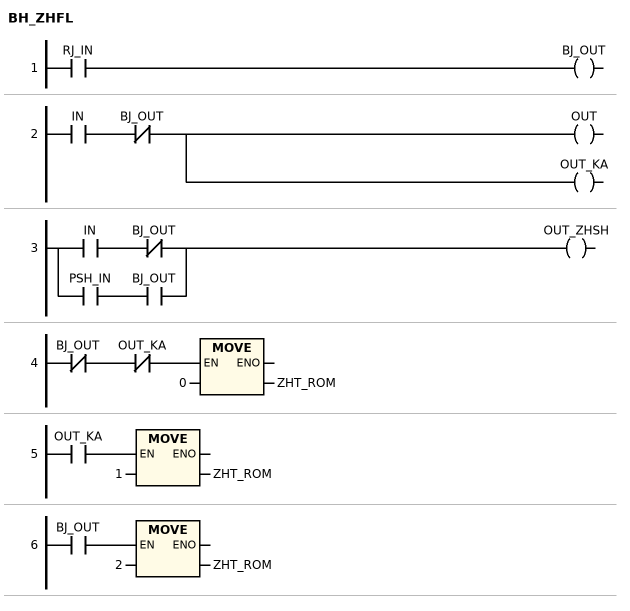
[picture p24: BH_ZHFL (LD)]
_LD_ (* Ladder Diagram *)
NETWORK 1
	[RJ_IN] --- (BJ_OUT)
NETWORK 2
	[IN] - [/BJ_OUT] --- (OUT) (OUT_KA)
NETWORK 3
	{ [IN] - [/BJ_OUT] | [PSH_IN] - [BJ_OUT] } --- (OUT_ZHSH)
NETWORK 4
	[/BJ_OUT] - [/OUT_KA]
		EN --- MOVE(0) => ZHT_ROM
NETWORK 5
	[OUT_KA]
		EN --- MOVE(1) => ZHT_ROM
NETWORK 6
	[BJ_OUT]
		EN --- MOVE(2) => ZHT_ROM
_END_LD_
(* the same logic as Structured Text *)
(* Network 1 *)
BJ_OUT := RJ_IN;
(* Network 2 *)
OUT := IN AND NOT BJ_OUT;
OUT_KA := OUT;
(* Network 3 *)
OUT_ZHSH := IN AND NOT BJ_OUT OR PSH_IN AND BJ_OUT;
(* Network 4 *)
IF NOT BJ_OUT AND NOT OUT_KA THEN
	ZHT_ROM := 0;
END_IF;
(* Network 5 *)
IF OUT_KA THEN
	ZHT_ROM := 1;
END_IF;
(* Network 6 *)
IF BJ_OUT THEN
	ZHT_ROM := 2;
END_IF;
END_FUNCTION_BLOCK

(* POU YOU_FEN, LD *)
FUNCTION_BLOCK YOU_FEN
VAR_INPUT
	MN_IN: INT;
	YW_XZH: INT;
	HIGH_IN: INT;
	LOW_IN: INT;
	YOU_WEI_IN: BOOL;
	TIME_IN: WORD;
	Y_LV_IN: BOOL;
	YL_SET: WORD;

	OPEN_IN: BOOL;
	RESET: BOOL;
	YF_IN: WORD;
	YF_XZ: INT;
END_VAR
VAR_OUTPUT
	YW_XH_OUT: INT;
	YL_KZH: BOOL;
	YOU_WEI_OUT: BOOL;
	TIME_OUT: WORD;
	YL_BJ: BOOL;
	YLV_XH: WORD;
	YL_PT: BOOL;
	YL_OUT: BOOL;
	YF_WD: INT;
	YF_JR: BOOL;
END_VAR
VAR
	TON_YW: YANSHI_OPEN;




	HIGH: BOOL;
	LOW: BOOL;
	KAIJI: BOOL;
	LIMITALARM: LIMITALARM;

	MID_KA: BOOL;
	YLV_YSH: YANSHI_OPEN;
	HYSTERESIS: HYSTERESIS;
	OUT: BOOL;
END_VAR
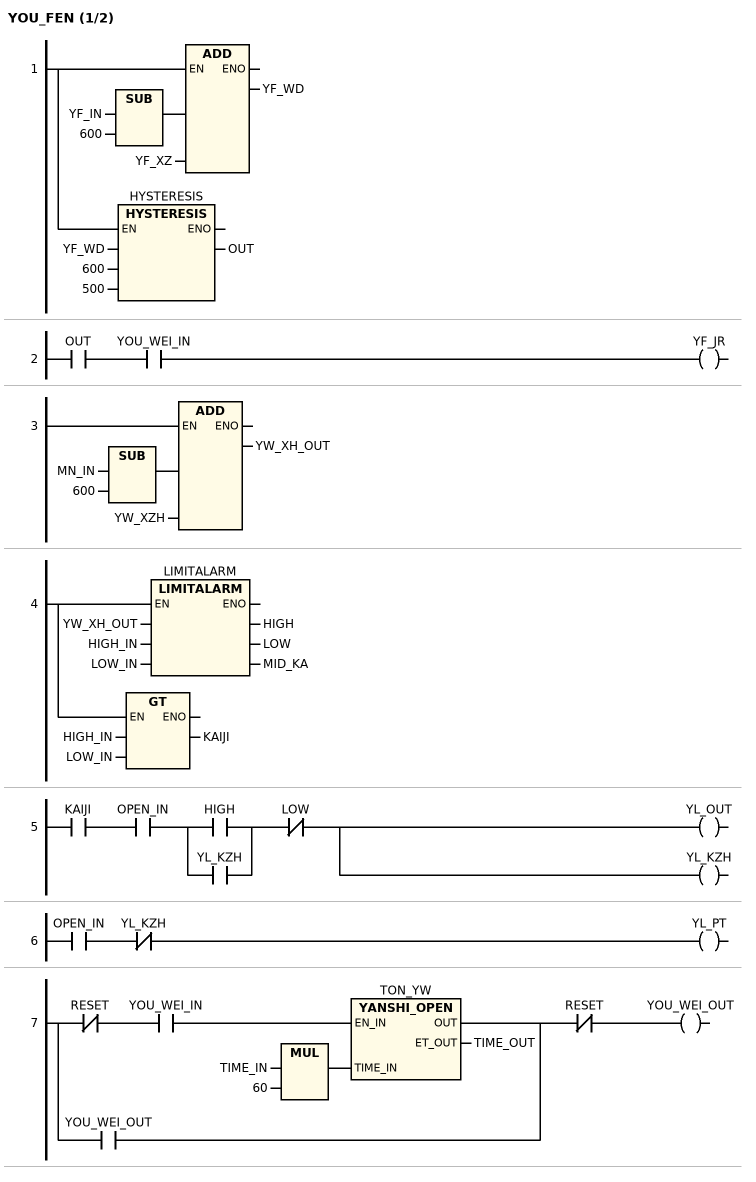
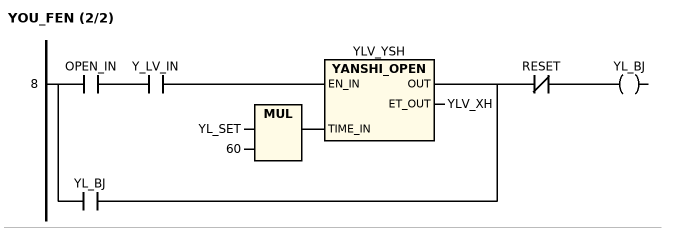
_LD_ (* Ladder Diagram *)
NETWORK 1
	*
		EN --- ADD(SUB(YF_IN, 600), YF_XZ) => YF_WD
		EN --- HYSTERESIS:HYSTERESIS(YF_WD, 600, 500) => OUT
NETWORK 2
	[OUT] - [YOU_WEI_IN] --- (YF_JR)
NETWORK 3
	*
		EN --- ADD(SUB(MN_IN, 600), YW_XZH) => YW_XH_OUT
NETWORK 4
	*
		EN --- LIMITALARM:LIMITALARM(YW_XH_OUT, HIGH_IN, LOW_IN, out 2 => LOW, out 3 => MID_KA) => HIGH
		EN --- GT(HIGH_IN, LOW_IN) => KAIJI
NETWORK 5
	[KAIJI] - [OPEN_IN] - { [HIGH] | [YL_KZH] } - [/LOW] --- (YL_OUT) (YL_KZH)
NETWORK 6
	[OPEN_IN] - [/YL_KZH] --- (YL_PT)
NETWORK 7
	{ [/RESET] - [YOU_WEI_IN] - TON_YW:YANSHI_OPEN(EN_IN: *, TIME_IN: MUL(TIME_IN, 60), ET_OUT => TIME_OUT) | [YOU_WEI_OUT] } - [/RESET] --- (YOU_WEI_OUT)
NETWORK 8
	{ [OPEN_IN] - [Y_LV_IN] - YLV_YSH:YANSHI_OPEN(EN_IN: *, TIME_IN: MUL(YL_SET, 60), ET_OUT => YLV_XH) | [YL_BJ] } - [/RESET] --- (YL_BJ)
_END_LD_
(* the same logic as Structured Text *)
(* Network 1: see the listing above *)
(* Network 2 *)
YF_JR := OUT AND YOU_WEI_IN;
(* Network 3 *)
YW_XH_OUT := (MN_IN - 600) + YW_XZH;
(* Network 4: see the listing above *)
(* Network 5 *)
YL_OUT := KAIJI AND OPEN_IN AND (HIGH OR YL_KZH) AND NOT LOW;
YL_KZH := YL_OUT;
(* Network 6 *)
YL_PT := OPEN_IN AND NOT YL_KZH;
(* Network 7 *)
TON_YW(EN_IN := NOT RESET AND YOU_WEI_IN, TIME_IN := TIME_IN * 60);
TIME_OUT := TON_YW.ET_OUT;
YOU_WEI_OUT := (TON_YW.OUT OR YOU_WEI_OUT) AND NOT RESET;
(* Network 8 *)
YLV_YSH(EN_IN := OPEN_IN AND Y_LV_IN, TIME_IN := YL_SET * 60);
YLV_XH := YLV_YSH.ET_OUT;
YL_BJ := (YLV_YSH.OUT OR YL_BJ) AND NOT RESET;
END_FUNCTION_BLOCK

(* POU SUO, LD *)
FUNCTION_BLOCK SUO
VAR_INPUT
	NIAN_IN: WORD;
	YUE_IN: WORD;
	RI_IN: WORD;
	NIAN_SET_1: WORD;
	YUE_SET_1: WORD;
	RI_SET_1: WORD;
	MIMA_1_IN: WORD;
	MIMA_1_SET_IN: WORD;
	NIAN_SET_2: WORD;
	YUE_SET_2: WORD;
	RI_SET_2: WORD;
	MIMA_2_IN: WORD;
	MIMA_2_SET_IN: WORD;

	NIAN_SET_3: WORD;
	YUE_SET_3: WORD;
	RI_SET_3: WORD;
	MIMA_3_IN: WORD;
	MIMA_3_SET_IN: WORD;
	OFF_ON: BOOL;


END_VAR
VAR_OUTPUT
	SUO_OUT: BOOL;
END_VAR
VAR
	SUO_NIAN_1: BOOL;
	SUO_YUE_1: BOOL;
	SUO_RI_1: BOOL;
	SUO_NIAN_2: BOOL;
	SUO_YUE_2: BOOL;
	SUO_RI_2: BOOL;
	SUO_NIAN_3: BOOL;
	SUO_YUE_3: BOOL;
	SUO_RI_3: BOOL;
	MIMA_1: BOOL;
	MIMA_2: BOOL;
	MIMA_3: BOOL;
	T_SUO_1: TON;
	T_SUO_2: TON;
	T_SUO_3: TON;
	TIME_SUO_1: TIME;
	TIME_SUO_2: TIME;
	TIME_SUO_3: TIME;
END_VAR
VAR_OUTPUT RETAIN
	SUO_1_OUT: BOOL;
	SUO_2_OUT: BOOL;
	SUO_3_OUT: BOOL;
END_VAR
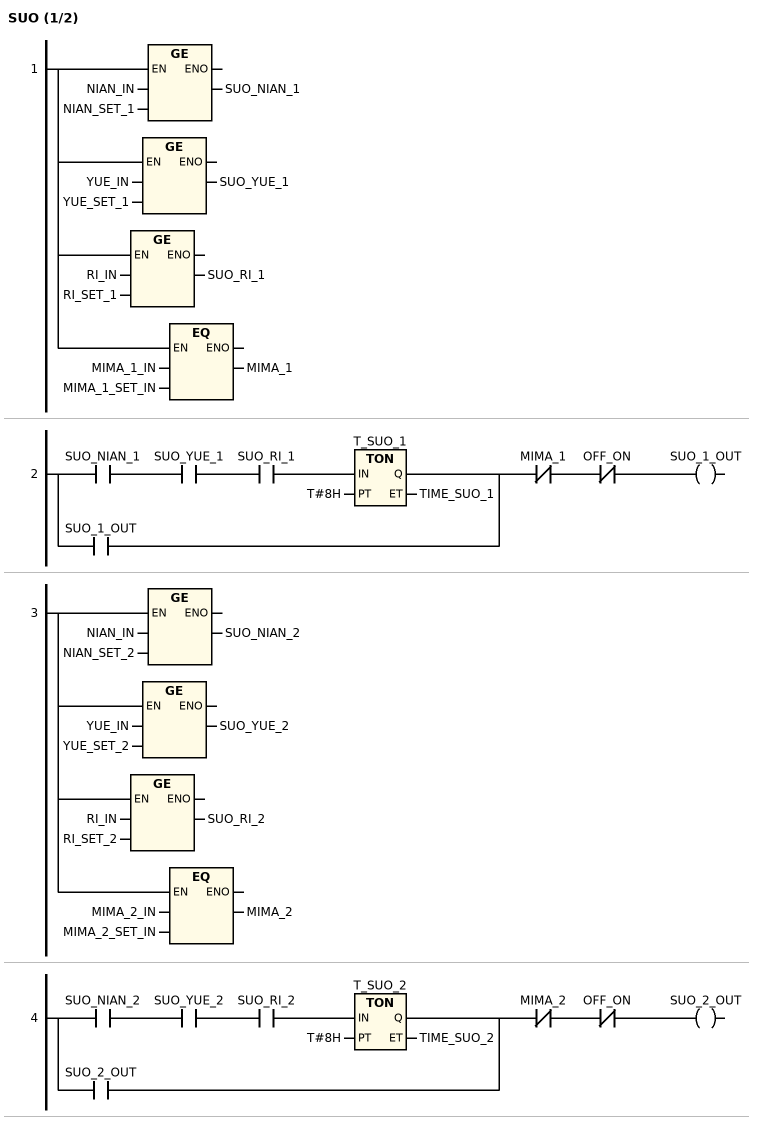
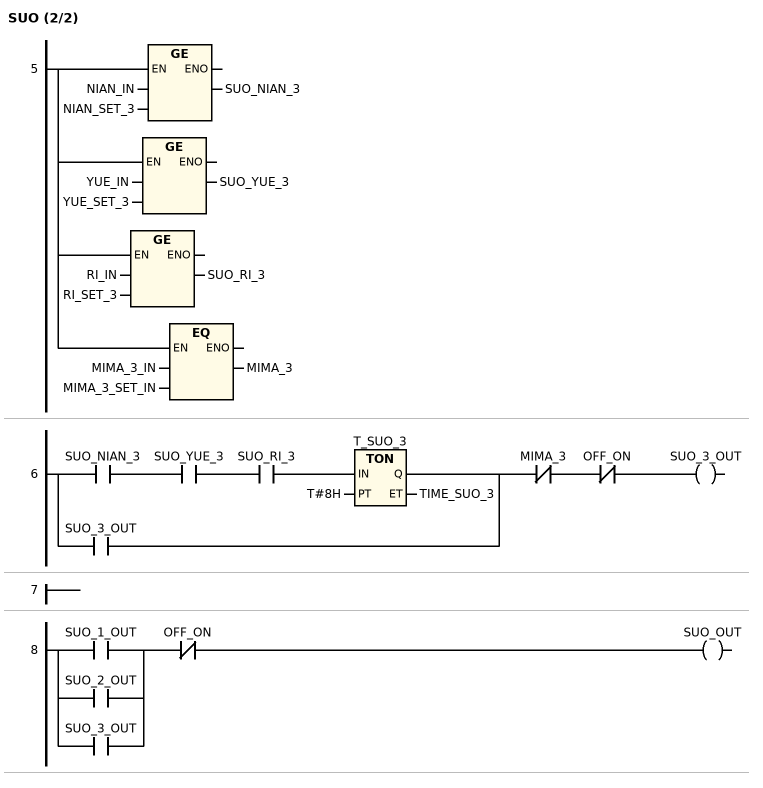
_LD_ (* Ladder Diagram *)
NETWORK 1
	*
		EN --- GE(NIAN_IN, NIAN_SET_1) => SUO_NIAN_1
		EN --- GE(YUE_IN, YUE_SET_1) => SUO_YUE_1
		EN --- GE(RI_IN, RI_SET_1) => SUO_RI_1
		EN --- EQ(MIMA_1_IN, MIMA_1_SET_IN) => MIMA_1
NETWORK 2
	{ [SUO_NIAN_1] - [SUO_YUE_1] - [SUO_RI_1] - T_SUO_1:TON(IN: *, PT: T#8H, ET => TIME_SUO_1) | [SUO_1_OUT] } - [/MIMA_1] - [/OFF_ON] --- (SUO_1_OUT)
NETWORK 3
	*
		EN --- GE(NIAN_IN, NIAN_SET_2) => SUO_NIAN_2
		EN --- GE(YUE_IN, YUE_SET_2) => SUO_YUE_2
		EN --- GE(RI_IN, RI_SET_2) => SUO_RI_2
		EN --- EQ(MIMA_2_IN, MIMA_2_SET_IN) => MIMA_2
NETWORK 4
	{ [SUO_NIAN_2] - [SUO_YUE_2] - [SUO_RI_2] - T_SUO_2:TON(IN: *, PT: T#8H, ET => TIME_SUO_2) | [SUO_2_OUT] } - [/MIMA_2] - [/OFF_ON] --- (SUO_2_OUT)
NETWORK 5
	*
		EN --- GE(NIAN_IN, NIAN_SET_3) => SUO_NIAN_3
		EN --- GE(YUE_IN, YUE_SET_3) => SUO_YUE_3
		EN --- GE(RI_IN, RI_SET_3) => SUO_RI_3
		EN --- EQ(MIMA_3_IN, MIMA_3_SET_IN) => MIMA_3
NETWORK 6
	{ [SUO_NIAN_3] - [SUO_YUE_3] - [SUO_RI_3] - T_SUO_3:TON(IN: *, PT: T#8H, ET => TIME_SUO_3) | [SUO_3_OUT] } - [/MIMA_3] - [/OFF_ON] --- (SUO_3_OUT)
NETWORK 7
	*
NETWORK 8
	{ [SUO_1_OUT] | [SUO_2_OUT] | [SUO_3_OUT] } - [/OFF_ON] --- (SUO_OUT)
_END_LD_
(* the same logic as Structured Text *)
(* Network 1 *)
SUO_NIAN_1 := NIAN_IN >= NIAN_SET_1;
SUO_YUE_1 := YUE_IN >= YUE_SET_1;
SUO_RI_1 := RI_IN >= RI_SET_1;
MIMA_1 := MIMA_1_IN = MIMA_1_SET_IN;
(* Network 2 *)
T_SUO_1(IN := SUO_NIAN_1 AND SUO_YUE_1 AND SUO_RI_1, PT := T#8H);
TIME_SUO_1 := T_SUO_1.ET;
SUO_1_OUT := (T_SUO_1.Q OR SUO_1_OUT) AND NOT MIMA_1 AND NOT OFF_ON;
(* Network 3 *)
SUO_NIAN_2 := NIAN_IN >= NIAN_SET_2;
SUO_YUE_2 := YUE_IN >= YUE_SET_2;
SUO_RI_2 := RI_IN >= RI_SET_2;
MIMA_2 := MIMA_2_IN = MIMA_2_SET_IN;
(* Network 4 *)
T_SUO_2(IN := SUO_NIAN_2 AND SUO_YUE_2 AND SUO_RI_2, PT := T#8H);
TIME_SUO_2 := T_SUO_2.ET;
SUO_2_OUT := (T_SUO_2.Q OR SUO_2_OUT) AND NOT MIMA_2 AND NOT OFF_ON;
(* Network 5 *)
SUO_NIAN_3 := NIAN_IN >= NIAN_SET_3;
SUO_YUE_3 := YUE_IN >= YUE_SET_3;
SUO_RI_3 := RI_IN >= RI_SET_3;
MIMA_3 := MIMA_3_IN = MIMA_3_SET_IN;
(* Network 6 *)
T_SUO_3(IN := SUO_NIAN_3 AND SUO_YUE_3 AND SUO_RI_3, PT := T#8H);
TIME_SUO_3 := T_SUO_3.ET;
SUO_3_OUT := (T_SUO_3.Q OR SUO_3_OUT) AND NOT MIMA_3 AND NOT OFF_ON;
(* Network 7 *)
(* Network 8 *)
SUO_OUT := (SUO_1_OUT OR SUO_2_OUT OR SUO_3_OUT) AND NOT OFF_ON;
END_FUNCTION_BLOCK

(* POU PQ_ZHFL_KZH, LD *)
FUNCTION_BLOCK PQ_ZHFL_KZH
VAR_INPUT
	OPEN_IN: BOOL;
	DY_IN: WORD;
	MNL_XZH: INT;
	DY_MU: INT;
	DY_MD: INT;
	MNL_HIGH_1_IN: INT;
	MNL_LOW_1_IN: INT;
	MNL_HIGH_2_IN: INT;
	MNL_LOW_2_IN: INT;
	MNL_HIGH_3_IN: INT;
	MNL_LOW_3_IN: INT;
	MNL_HIGH_4_IN: INT;
	MNL_LOW_4_IN: INT;
	MNL_HIGH_SHB_IN: INT;
	MNL_LOW_SHB_IN: INT;
	MNL_HIGH_SHB2_IN: INT;
	MNL_LOW_SHB2_IN: INT;
	GY_IN: BOOL;
	LN_AN: BOOL;

	XH_JG: WORD;
	XH_SC: WORD;
	DXJ: BOOL;
	YA_IN: WORD;
	SET_YA: INT;
END_VAR
VAR_OUTPUT
	MNL_OUT: INT;
	FAN_1_OUT: BOOL;
	FAN_2_OUT: BOOL;
	FAN_3_OUT: BOOL;
	FAN_4_OUT: BOOL;
	SHB_OUT: BOOL;
	SHB2_OUT: BOOL;
	LN_NIU: BOOL;
	YOU_YA: INT;
	YA_CHA: INT;
	YA_BJ: BOOL;
END_VAR
VAR
	MNL_R: REAL;
	DIYA: HEX_ENGIN;





	MN_FAN_1: LIMITALARM;
	HIGH_1: BOOL;
	LOW_1: BOOL;
	MID_1: BOOL;
	KAIJI_1: BOOL;
	MN_FAN_2: LIMITALARM;
	HIGH_2: BOOL;
	LOW_2: BOOL;
	MID_2: BOOL;
	KAIJI_2: BOOL;
	MN_FAN_3: LIMITALARM;
	HIGH_3: BOOL;
	LOW_3: BOOL;
	MID_3: BOOL;
	KAIJI_3: BOOL;
	MN_FAN_4: LIMITALARM;
	HIGH_4: BOOL;
	LOW_4: BOOL;
	MID_4: BOOL;
	KAIJI_4: BOOL;
	MN_SHB: LIMITALARM;
	HIGH_SHB: BOOL;
	LOW_SHB: BOOL;
	MID_SHB: BOOL;
	KAIJI_SHB: BOOL;
	MN_SHB2: LIMITALARM;
	HIGH_SHB2: BOOL;
	LOW_SHB2: BOOL;
	MID_SHB2: BOOL;
	KAIJI_SHB2: BOOL;
	ZHFL_KZH: BOOL;
	LN_KZH: AN_NIU;

	BLINK: BLINK;
	DJ_K: BOOL;
	JG_O: BOOL;
	SC_O: BOOL;
	HEX_E: HEX_ENGIN;
END_VAR
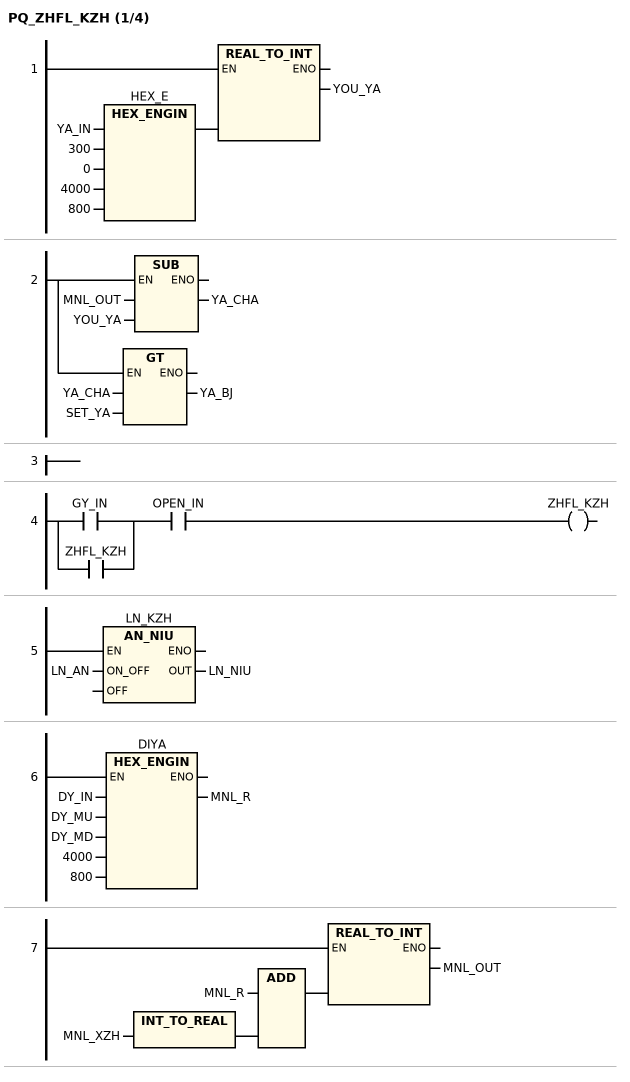
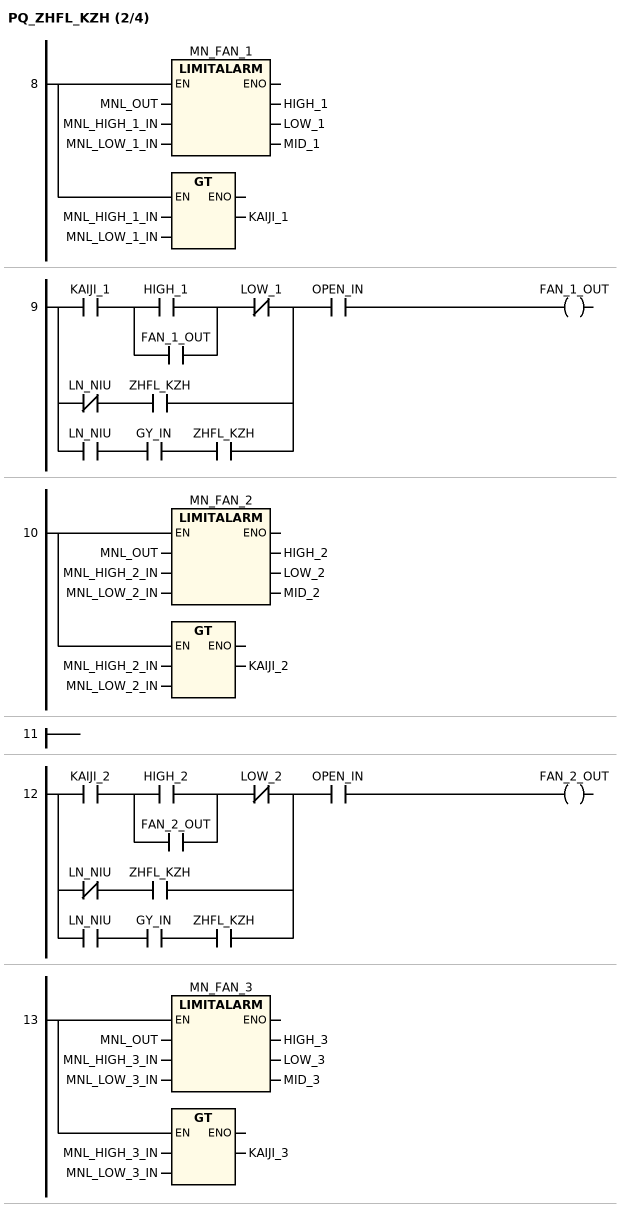
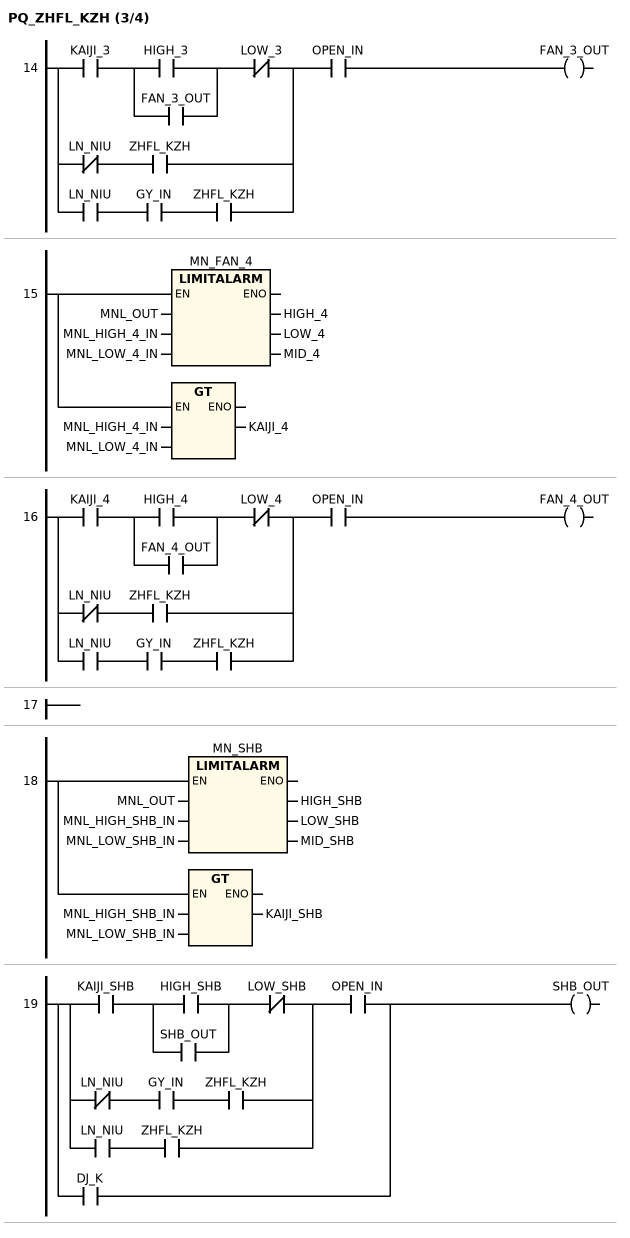
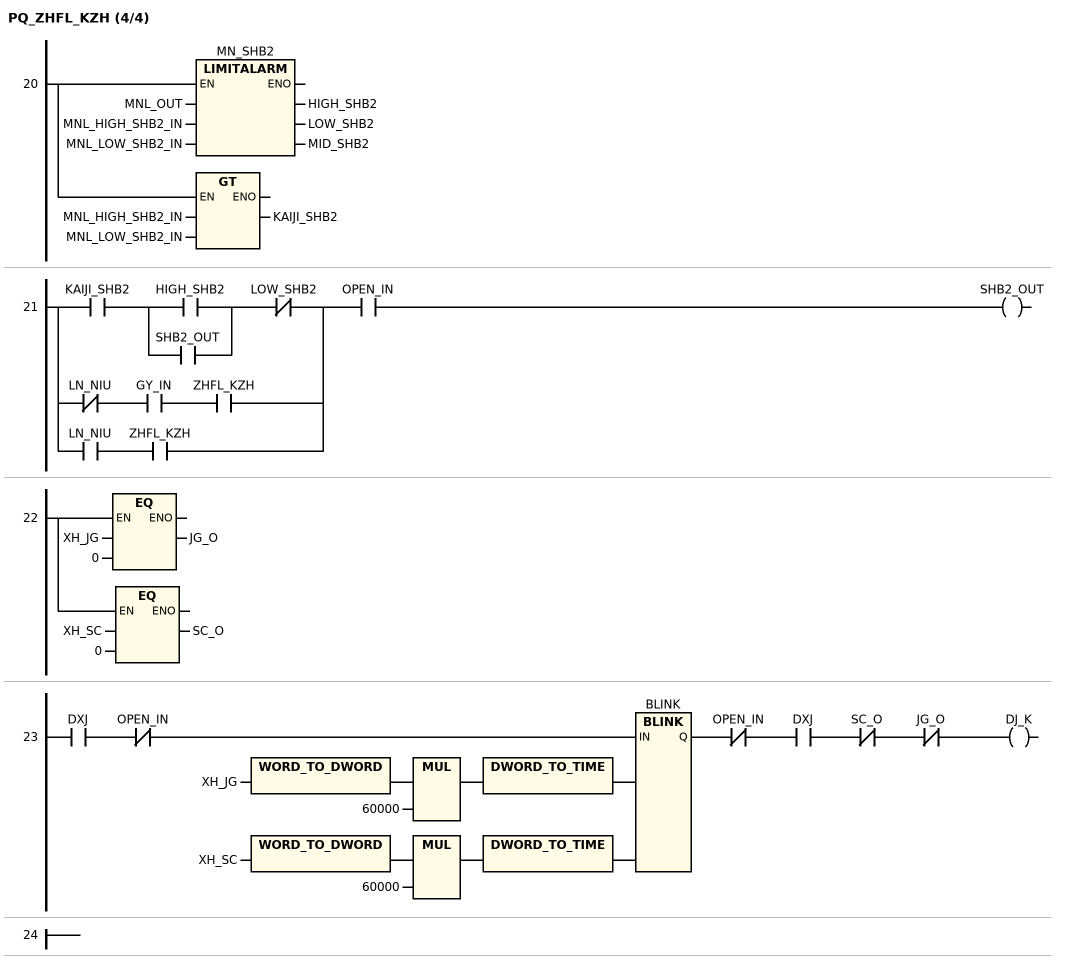
_LD_ (* Ladder Diagram *)
NETWORK 1
	*
		EN --- REAL_TO_INT(HEX_E:HEX_ENGIN(YA_IN, 300, 0, 4000, 800)) => YOU_YA
NETWORK 2
	*
		EN --- SUB(MNL_OUT, YOU_YA) => YA_CHA
		EN --- GT(YA_CHA, SET_YA) => YA_BJ
NETWORK 3
	*
NETWORK 4
	{ [GY_IN] | [ZHFL_KZH] } - [OPEN_IN] --- (ZHFL_KZH)
NETWORK 5
	*
		EN --- LN_KZH:AN_NIU(ON_OFF: LN_AN, OFF: ) => LN_NIU
NETWORK 6
	*
		EN --- DIYA:HEX_ENGIN(DY_IN, DY_MU, DY_MD, 4000, 800) => MNL_R
NETWORK 7
	*
		EN --- REAL_TO_INT(ADD(MNL_R, INT_TO_REAL(MNL_XZH))) => MNL_OUT
NETWORK 8
	*
		EN --- MN_FAN_1:LIMITALARM(MNL_OUT, MNL_HIGH_1_IN, MNL_LOW_1_IN, out 2 => LOW_1, out 3 => MID_1) => HIGH_1
		EN --- GT(MNL_HIGH_1_IN, MNL_LOW_1_IN) => KAIJI_1
NETWORK 9
	{ [KAIJI_1] - { [HIGH_1] | [FAN_1_OUT] } - [/LOW_1] | [/LN_NIU] - [ZHFL_KZH] | [LN_NIU] - [GY_IN] - [ZHFL_KZH] } - [OPEN_IN] --- (FAN_1_OUT)
NETWORK 10
	*
		EN --- MN_FAN_2:LIMITALARM(MNL_OUT, MNL_HIGH_2_IN, MNL_LOW_2_IN, out 2 => LOW_2, out 3 => MID_2) => HIGH_2
		EN --- GT(MNL_HIGH_2_IN, MNL_LOW_2_IN) => KAIJI_2
NETWORK 11
	*
NETWORK 12
	{ [KAIJI_2] - { [HIGH_2] | [FAN_2_OUT] } - [/LOW_2] | [/LN_NIU] - [ZHFL_KZH] | [LN_NIU] - [GY_IN] - [ZHFL_KZH] } - [OPEN_IN] --- (FAN_2_OUT)
NETWORK 13
	*
		EN --- MN_FAN_3:LIMITALARM(MNL_OUT, MNL_HIGH_3_IN, MNL_LOW_3_IN, out 2 => LOW_3, out 3 => MID_3) => HIGH_3
		EN --- GT(MNL_HIGH_3_IN, MNL_LOW_3_IN) => KAIJI_3
NETWORK 14
	{ [KAIJI_3] - { [HIGH_3] | [FAN_3_OUT] } - [/LOW_3] | [/LN_NIU] - [ZHFL_KZH] | [LN_NIU] - [GY_IN] - [ZHFL_KZH] } - [OPEN_IN] --- (FAN_3_OUT)
NETWORK 15
	*
		EN --- MN_FAN_4:LIMITALARM(MNL_OUT, MNL_HIGH_4_IN, MNL_LOW_4_IN, out 2 => LOW_4, out 3 => MID_4) => HIGH_4
		EN --- GT(MNL_HIGH_4_IN, MNL_LOW_4_IN) => KAIJI_4
NETWORK 16
	{ [KAIJI_4] - { [HIGH_4] | [FAN_4_OUT] } - [/LOW_4] | [/LN_NIU] - [ZHFL_KZH] | [LN_NIU] - [GY_IN] - [ZHFL_KZH] } - [OPEN_IN] --- (FAN_4_OUT)
NETWORK 17
	*
NETWORK 18
	*
		EN --- MN_SHB:LIMITALARM(MNL_OUT, MNL_HIGH_SHB_IN, MNL_LOW_SHB_IN, out 2 => LOW_SHB, out 3 => MID_SHB) => HIGH_SHB
		EN --- GT(MNL_HIGH_SHB_IN, MNL_LOW_SHB_IN) => KAIJI_SHB
NETWORK 19
	{ { [KAIJI_SHB] - { [HIGH_SHB] | [SHB_OUT] } - [/LOW_SHB] | [/LN_NIU] - [GY_IN] - [ZHFL_KZH] | [LN_NIU] - [ZHFL_KZH] } - [OPEN_IN] | [DJ_K] } --- (SHB_OUT)
NETWORK 20
	*
		EN --- MN_SHB2:LIMITALARM(MNL_OUT, MNL_HIGH_SHB2_IN, MNL_LOW_SHB2_IN, out 2 => LOW_SHB2, out 3 => MID_SHB2) => HIGH_SHB2
		EN --- GT(MNL_HIGH_SHB2_IN, MNL_LOW_SHB2_IN) => KAIJI_SHB2
NETWORK 21
	{ [KAIJI_SHB2] - { [HIGH_SHB2] | [SHB2_OUT] } - [/LOW_SHB2] | [/LN_NIU] - [GY_IN] - [ZHFL_KZH] | [LN_NIU] - [ZHFL_KZH] } - [OPEN_IN] --- (SHB2_OUT)
NETWORK 22
	*
		EN --- EQ(XH_JG, 0) => JG_O
		EN --- EQ(XH_SC, 0) => SC_O
NETWORK 23
	[DXJ] - [/OPEN_IN] - BLINK:BLINK(*, DWORD_TO_TIME(MUL(WORD_TO_DWORD(XH_JG), 60000)), DWORD_TO_TIME(MUL(WORD_TO_DWORD(XH_SC), 60000))) - [/OPEN_IN] - [DXJ] - [/SC_O] - [/JG_O] --- (DJ_K)
NETWORK 24
	*
_END_LD_
(* the same logic as Structured Text *)
(* Network 1: see the listing above *)
(* Network 2 *)
YA_CHA := MNL_OUT - YOU_YA;
YA_BJ := YA_CHA > SET_YA;
(* Network 3: see the listing above *)
(* Network 4 *)
ZHFL_KZH := (GY_IN OR ZHFL_KZH) AND OPEN_IN;
(* Network 5: see the listing above *)
(* Network 6: see the listing above *)
(* Network 7 *)
MNL_OUT := REAL_TO_INT(MNL_R + INT_TO_REAL(MNL_XZH));
(* Network 8: see the listing above *)
(* Network 9 *)
FAN_1_OUT := (KAIJI_1 AND (HIGH_1 OR FAN_1_OUT) AND NOT LOW_1 OR NOT LN_NIU AND ZHFL_KZH OR LN_NIU AND GY_IN AND ZHFL_KZH) AND OPEN_IN;
(* Network 10: see the listing above *)
(* Network 11: see the listing above *)
(* Network 12 *)
FAN_2_OUT := (KAIJI_2 AND (HIGH_2 OR FAN_2_OUT) AND NOT LOW_2 OR NOT LN_NIU AND ZHFL_KZH OR LN_NIU AND GY_IN AND ZHFL_KZH) AND OPEN_IN;
(* Network 13: see the listing above *)
(* Network 14 *)
FAN_3_OUT := (KAIJI_3 AND (HIGH_3 OR FAN_3_OUT) AND NOT LOW_3 OR NOT LN_NIU AND ZHFL_KZH OR LN_NIU AND GY_IN AND ZHFL_KZH) AND OPEN_IN;
(* Network 15: see the listing above *)
(* Network 16 *)
FAN_4_OUT := (KAIJI_4 AND (HIGH_4 OR FAN_4_OUT) AND NOT LOW_4 OR NOT LN_NIU AND ZHFL_KZH OR LN_NIU AND GY_IN AND ZHFL_KZH) AND OPEN_IN;
(* Network 17: see the listing above *)
(* Network 18: see the listing above *)
(* Network 19 *)
SHB_OUT := (KAIJI_SHB AND (HIGH_SHB OR SHB_OUT) AND NOT LOW_SHB OR NOT LN_NIU AND GY_IN AND ZHFL_KZH OR LN_NIU AND ZHFL_KZH) AND OPEN_IN OR DJ_K;
(* Network 20: see the listing above *)
(* Network 21 *)
SHB2_OUT := (KAIJI_SHB2 AND (HIGH_SHB2 OR SHB2_OUT) AND NOT LOW_SHB2 OR NOT LN_NIU AND GY_IN AND ZHFL_KZH OR LN_NIU AND ZHFL_KZH) AND OPEN_IN;
(* Network 22 *)
JG_O := XH_JG = 0;
SC_O := XH_SC = 0;
(* Network 23: see the listing above *)
(* Network 24: see the listing above *)
END_FUNCTION_BLOCK

(* POU AN_NIU, LD *)
FUNCTION_BLOCK AN_NIU
VAR_INPUT
	ON_OFF: BOOL;
	OFF: BOOL;
END_VAR
VAR_OUTPUT
       END_VAR
VAR
	R1: R_TRIG;
	R1_Q: BOOL;
END_VAR
VAR_OUTPUT RETAIN
	OUT: BOOL;
END_VAR
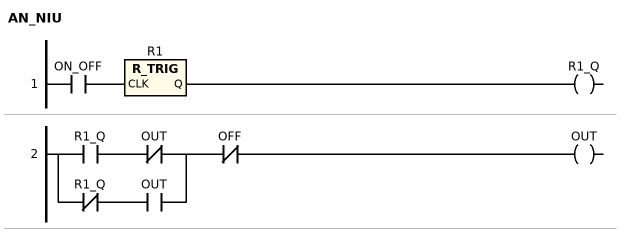
_LD_ (* Ladder Diagram *)
NETWORK 1
	[ON_OFF] - R1:R_TRIG(CLK: *) --- (R1_Q)
NETWORK 2
	{ [R1_Q] - [/OUT] | [/R1_Q] - [OUT] } - [/OFF] --- (OUT)
_END_LD_
(* the same logic as Structured Text *)
(* Network 1 *)
R1(CLK := ON_OFF);
R1_Q := R1.Q;
(* Network 2 *)
OUT := (R1_Q AND NOT OUT OR NOT R1_Q AND OUT) AND NOT OFF;
END_FUNCTION_BLOCK

(* POU XH_YANSHI_1, LD *)
FUNCTION_BLOCK XH_YANSHI_1
VAR_INPUT
	WBKZL_IN: BOOL;
	OPEN_IN: BOOL;
	DY_IN: WORD;
	MNL_XZH: INT;
	MNL_HIGH_IN: INT;
	MNL_LOW_IN: INT;
	OPEN_YSH: WORD;
	CLOSE_YSH: WORD;
	JQ_OPEN_YSH: WORD;
 	JQ_1_BH_IN: BOOL;
	JQ_2_BH_IN: BOOL;
	JQ_3_BH_IN: BOOL;
	JQ_4_BH_IN: BOOL;
	JQ_5_BH_IN: BOOL;
	JQ_6_BH_IN: BOOL;


	DY_MU: INT;
	DY_MD: INT;
	JQ_NJ_SHU: WORD;
	WD_IN: WORD;
	XQ_WD_XZH: INT;
	WD_MU: INT;
	WD_MD: INT;
	GRD_IN: INT;
	GRD_YSH_SET: WORD;
	TD_R: BOOL;
	TJ_ZHH: BOOL;

	YSJ_IN: BOOL;
	RESET: BOOL;
END_VAR
VAR_OUTPUT
	MNL_OUT: INT;
	YL_T_OUT: INT;
	XH_T_XSH: WORD;
	XH_SHU_OUT: WORD;
	XH_ZHT: WORD;


	JJQ_OUT: BOOL;
	XQ_WD_OUT: INT;
	GRD_OUT: INT;
	GRD_ALA: BOOL;
	GRD_YSH_XSH: WORD;
	TJ_ZHH_OUT: BOOL;
END_VAR
VAR
	HIGH: BOOL;
	MID: BOOL;
	CLOSE_SET: TIME;
	OPEN_SET: TIME;
	JQ_OPEN_SET: TIME;
	H_R_Q: BOOL;
	H_TON: TON;
	JT_TON: TON;
	JT_KA: BOOL;
	XH_JD: BOOL;
	JT_SHU: WORD;
	XH_STOP: BOOL;
	XH_NE_3: BOOL;
	JQ_A_OPEN_SET_0: BOOL;
	LOW_R: R_TRIG;
	LOW_R_Q: BOOL;
	L_R_Q: BOOL;
	L_TON: TON;
	XH_SHU_0: BOOL;
	JQ_OPEN_SET_0: BOOL;
	LOW: BOOL;
	XH_NE_6: BOOL;
	XH_NE_12: BOOL;
	XH_NE_18: BOOL;
	XH_EQ_3: BOOL;
	XH_EQ_6: BOOL;
	XH_EQ_9: BOOL;
	XH_EQ_12: BOOL;
	XH_EQ_15: BOOL;
	XH_EQ_18: BOOL;
	HIG_R: R_TRIG;
	XH_NE_9: BOOL;
	MNL_R: REAL;
	MONI_LIANG: LIMITALARM;
	HIGH_KA: BOOL;
	LOW_KA: BOOL;
	MID_KA: BOOL;
	KAIJI: BOOL;
	XH_SHU: WORD;
	OPEN_ET: TIME;
	CLOSE_ET: TIME;
	JT_OPEN_ET: TIME;
	XH_JT_KA: BOOL;
	HIG_KA_R: R_TRIG;
	DIYA: HEX_ENGIN;
	YL_WD: YL_WD;



	MID_R: R_TRIG;


	GRD_KA: BOOL;
	GRD_OPEN: YANSHI_OPEN;
	GRD_KA_0: BOOL;
	JQ_NJ_SHU_0: BOOL;
	JJQ_TOF: TOF;
	TJ_AN: AN_NIU;
	HEX_ENGIN: HEX_ENGIN;
	wd: HEX_ENGIN;
	HEX_ENGI: HEX_ENGIN;
	XW: INT;
END_VAR
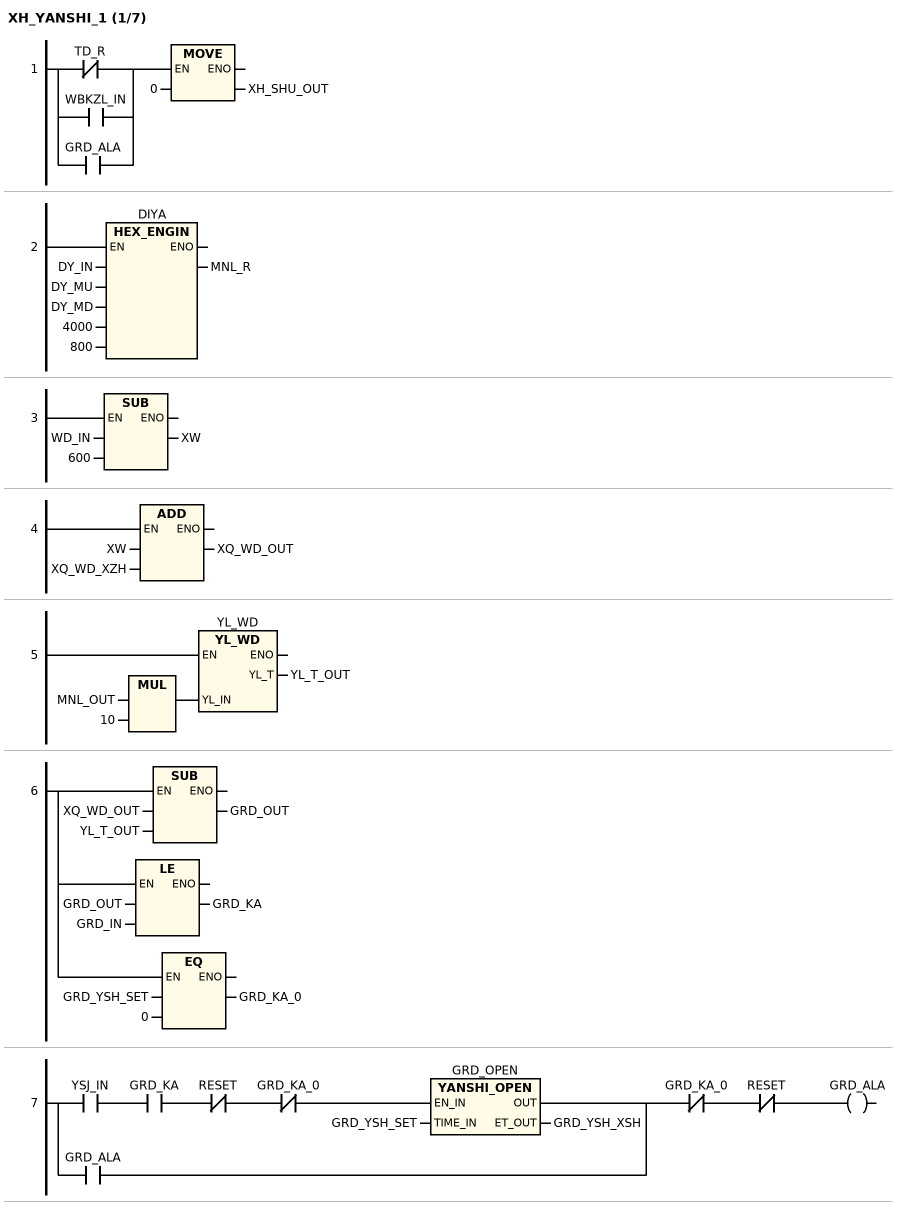
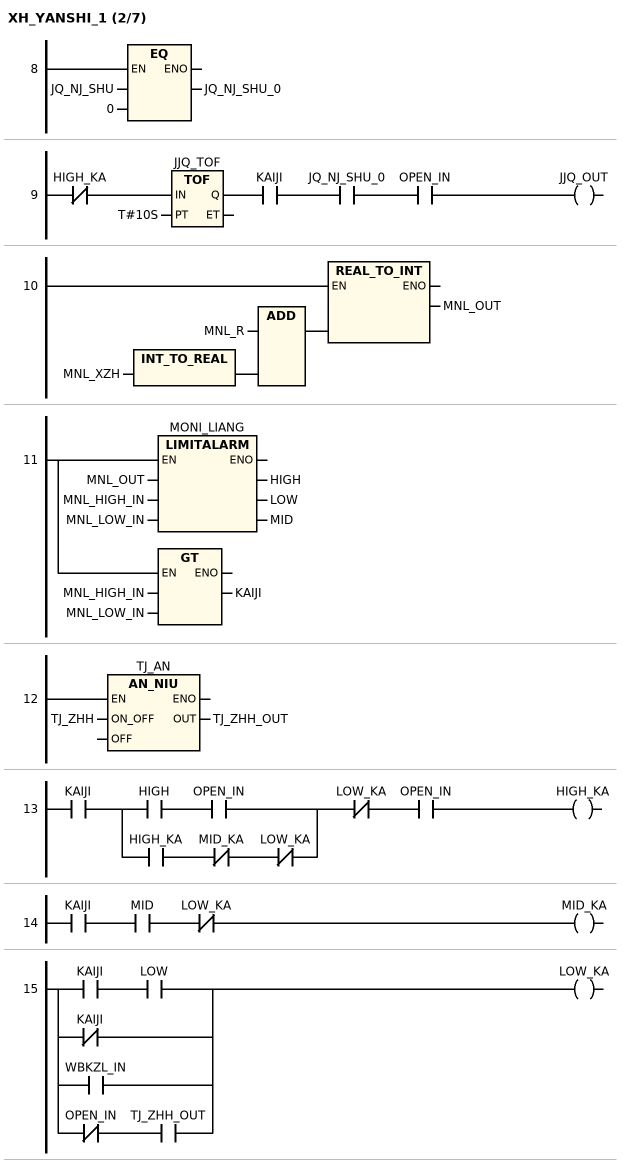
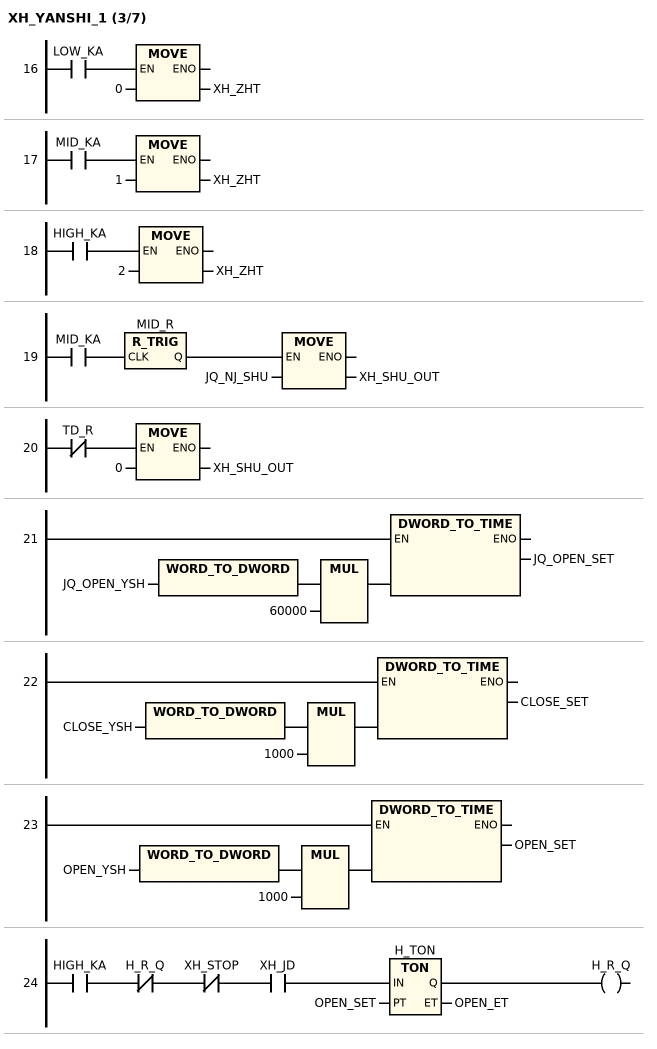
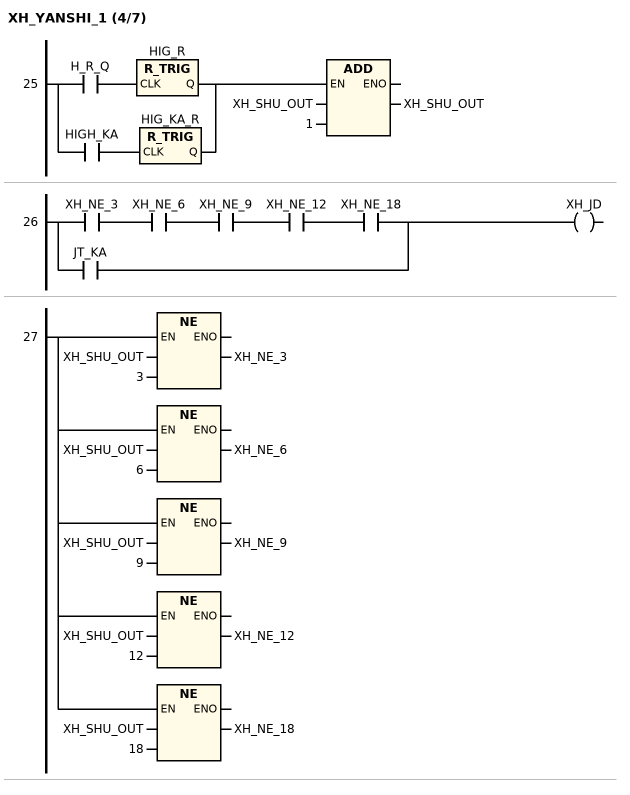
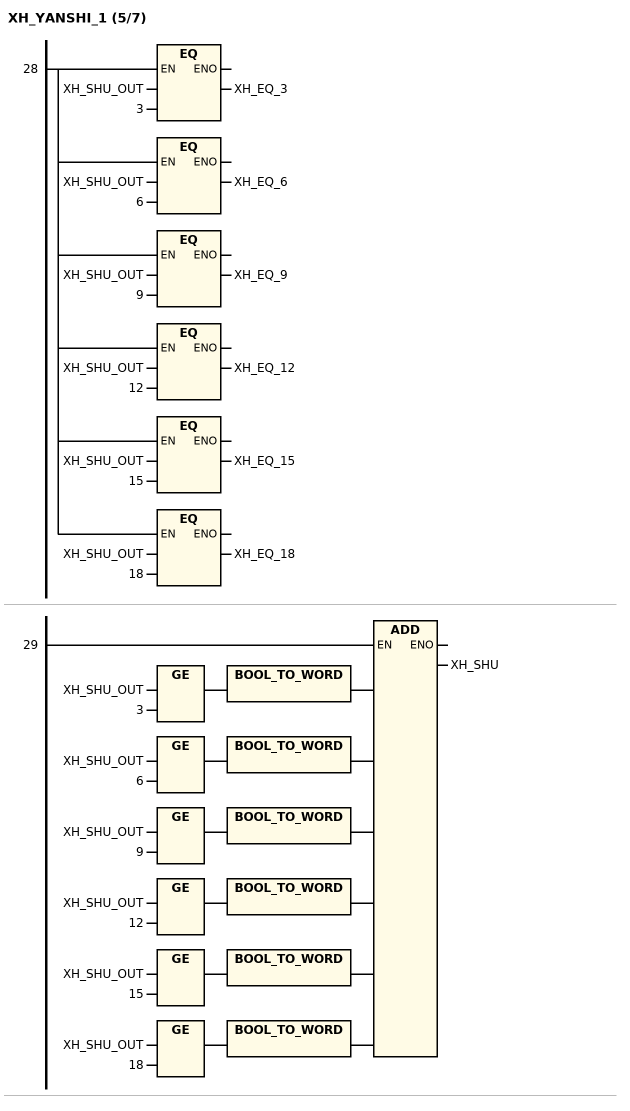
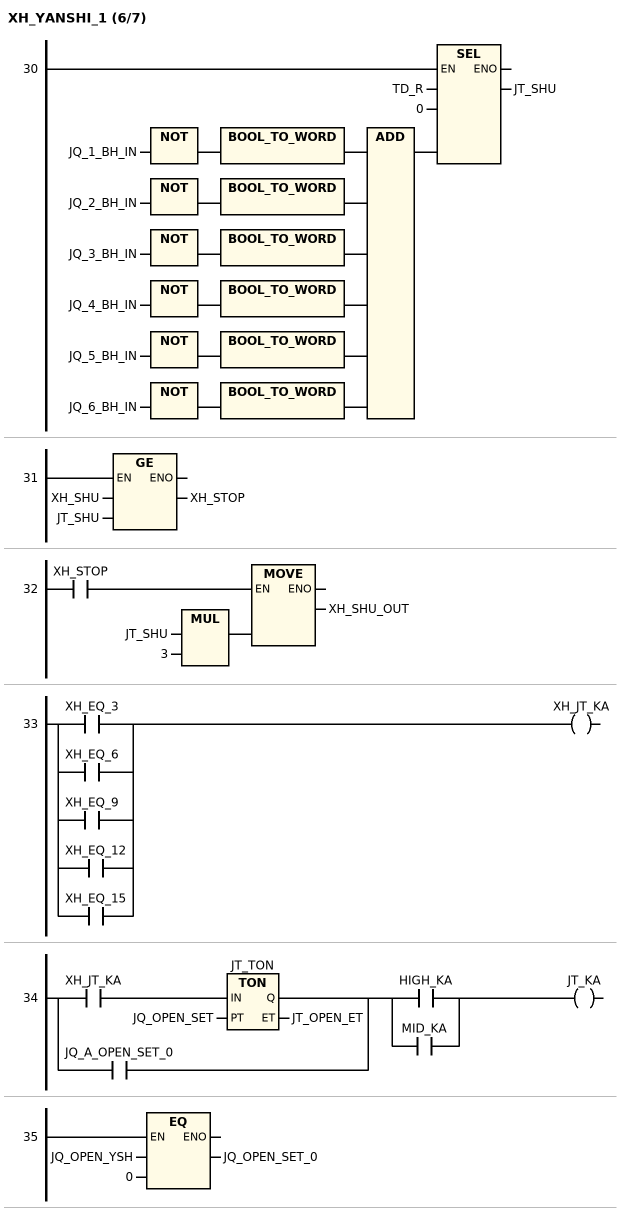
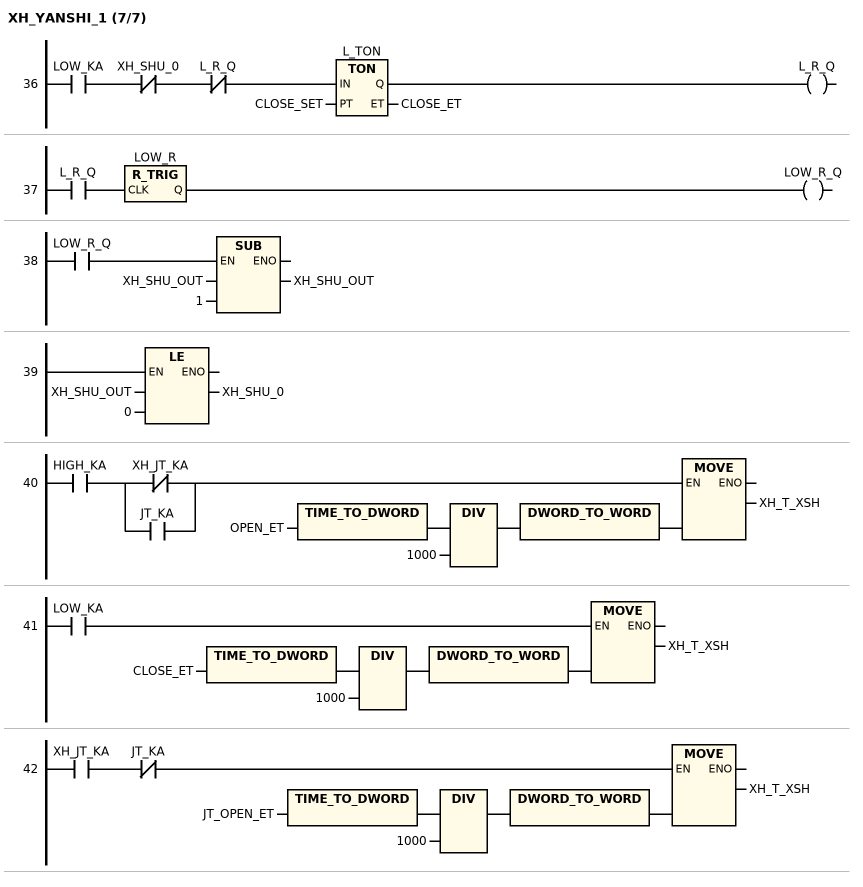
_LD_ (* Ladder Diagram *)
NETWORK 1
	{ [/TD_R] | [WBKZL_IN] | [GRD_ALA] }
		EN --- MOVE(0) => XH_SHU_OUT
NETWORK 2
	*
		EN --- DIYA:HEX_ENGIN(DY_IN, DY_MU, DY_MD, 4000, 800) => MNL_R
NETWORK 3
	*
		EN --- SUB(WD_IN, 600) => XW
NETWORK 4
	*
		EN --- ADD(XW, XQ_WD_XZH) => XQ_WD_OUT
NETWORK 5
	*
		EN --- YL_WD:YL_WD(YL_IN: MUL(MNL_OUT, 10)) => YL_T_OUT
NETWORK 6
	*
		EN --- SUB(XQ_WD_OUT, YL_T_OUT) => GRD_OUT
		EN --- LE(GRD_OUT, GRD_IN) => GRD_KA
		EN --- EQ(GRD_YSH_SET, 0) => GRD_KA_0
NETWORK 7
	{ [YSJ_IN] - [GRD_KA] - [/RESET] - [/GRD_KA_0] - GRD_OPEN:YANSHI_OPEN(EN_IN: *, TIME_IN: GRD_YSH_SET, ET_OUT => GRD_YSH_XSH) | [GRD_ALA] } - [/GRD_KA_0] - [/RESET] --- (GRD_ALA)
NETWORK 8
	*
		EN --- EQ(JQ_NJ_SHU, 0) => JQ_NJ_SHU_0
NETWORK 9
	[/HIGH_KA] - JJQ_TOF:TOF(IN: *, PT: T#10S) - [KAIJI] - [JQ_NJ_SHU_0] - [OPEN_IN] --- (JJQ_OUT)
NETWORK 10
	*
		EN --- REAL_TO_INT(ADD(MNL_R, INT_TO_REAL(MNL_XZH))) => MNL_OUT
NETWORK 11
	*
		EN --- MONI_LIANG:LIMITALARM(MNL_OUT, MNL_HIGH_IN, MNL_LOW_IN, out 2 => LOW, out 3 => MID) => HIGH
		EN --- GT(MNL_HIGH_IN, MNL_LOW_IN) => KAIJI
NETWORK 12
	*
		EN --- TJ_AN:AN_NIU(ON_OFF: TJ_ZHH, OFF: ) => TJ_ZHH_OUT
NETWORK 13
	[KAIJI] - { [HIGH] - [OPEN_IN] | [HIGH_KA] - [/MID_KA] - [/LOW_KA] } - [/LOW_KA] - [OPEN_IN] --- (HIGH_KA)
NETWORK 14
	[KAIJI] - [MID] - [/LOW_KA] --- (MID_KA)
NETWORK 15
	{ [KAIJI] - [LOW] | [/KAIJI] | [WBKZL_IN] | [/OPEN_IN] - [TJ_ZHH_OUT] } --- (LOW_KA)
NETWORK 16
	[LOW_KA]
		EN --- MOVE(0) => XH_ZHT
NETWORK 17
	[MID_KA]
		EN --- MOVE(1) => XH_ZHT
NETWORK 18
	[HIGH_KA]
		EN --- MOVE(2) => XH_ZHT
NETWORK 19
	[MID_KA] - MID_R:R_TRIG(CLK: *)
		EN --- MOVE(JQ_NJ_SHU) => XH_SHU_OUT
NETWORK 20
	[/TD_R]
		EN --- MOVE(0) => XH_SHU_OUT
NETWORK 21
	*
		EN --- DWORD_TO_TIME(MUL(WORD_TO_DWORD(JQ_OPEN_YSH), 60000)) => JQ_OPEN_SET
NETWORK 22
	*
		EN --- DWORD_TO_TIME(MUL(WORD_TO_DWORD(CLOSE_YSH), 1000)) => CLOSE_SET
NETWORK 23
	*
		EN --- DWORD_TO_TIME(MUL(WORD_TO_DWORD(OPEN_YSH), 1000)) => OPEN_SET
NETWORK 24
	[HIGH_KA] - [/H_R_Q] - [/XH_STOP] - [XH_JD] - H_TON:TON(IN: *, PT: OPEN_SET, ET => OPEN_ET) --- (H_R_Q)
NETWORK 25
	{ [H_R_Q] - HIG_R:R_TRIG(CLK: *) | [HIGH_KA] - HIG_KA_R:R_TRIG(CLK: *) }
		EN --- ADD(XH_SHU_OUT, 1) => XH_SHU_OUT
NETWORK 26
	{ [XH_NE_3] - [XH_NE_6] - [XH_NE_9] - [XH_NE_12] - [XH_NE_18] | [JT_KA] } --- (XH_JD)
NETWORK 27
	*
		EN --- NE(XH_SHU_OUT, 3) => XH_NE_3
		EN --- NE(XH_SHU_OUT, 6) => XH_NE_6
		EN --- NE(XH_SHU_OUT, 9) => XH_NE_9
		EN --- NE(XH_SHU_OUT, 12) => XH_NE_12
		EN --- NE(XH_SHU_OUT, 18) => XH_NE_18
NETWORK 28
	*
		EN --- EQ(XH_SHU_OUT, 3) => XH_EQ_3
		EN --- EQ(XH_SHU_OUT, 6) => XH_EQ_6
		EN --- EQ(XH_SHU_OUT, 9) => XH_EQ_9
		EN --- EQ(XH_SHU_OUT, 12) => XH_EQ_12
		EN --- EQ(XH_SHU_OUT, 15) => XH_EQ_15
		EN --- EQ(XH_SHU_OUT, 18) => XH_EQ_18
NETWORK 29
	*
		EN --- ADD(BOOL_TO_WORD(GE(XH_SHU_OUT, 3)), BOOL_TO_WORD(GE(XH_SHU_OUT, 6)), BOOL_TO_WORD(GE(XH_SHU_OUT, 9)), BOOL_TO_WORD(GE(XH_SHU_OUT, 12)), BOOL_TO_WORD(GE(XH_SHU_OUT, 15)), BOOL_TO_WORD(GE(XH_SHU_OUT, 18))) => XH_SHU
NETWORK 30
	*
		EN --- SEL(TD_R, 0, ADD(BOOL_TO_WORD(NOT(JQ_1_BH_IN)), BOOL_TO_WORD(NOT(JQ_2_BH_IN)), BOOL_TO_WORD(NOT(JQ_3_BH_IN)), BOOL_TO_WORD(NOT(JQ_4_BH_IN)), BOOL_TO_WORD(NOT(JQ_5_BH_IN)), BOOL_TO_WORD(NOT(JQ_6_BH_IN)))) => JT_SHU
NETWORK 31
	*
		EN --- GE(XH_SHU, JT_SHU) => XH_STOP
NETWORK 32
	[XH_STOP]
		EN --- MOVE(MUL(JT_SHU, 3)) => XH_SHU_OUT
NETWORK 33
	{ [XH_EQ_3] | [XH_EQ_6] | [XH_EQ_9] | [XH_EQ_12] | [XH_EQ_15] } --- (XH_JT_KA)
NETWORK 34
	{ [XH_JT_KA] - JT_TON:TON(IN: *, PT: JQ_OPEN_SET, ET => JT_OPEN_ET) | [JQ_A_OPEN_SET_0] } - { [HIGH_KA] | [MID_KA] } --- (JT_KA)
NETWORK 35
	*
		EN --- EQ(JQ_OPEN_YSH, 0) => JQ_OPEN_SET_0
NETWORK 36
	[LOW_KA] - [/XH_SHU_0] - [/L_R_Q] - L_TON:TON(IN: *, PT: CLOSE_SET, ET => CLOSE_ET) --- (L_R_Q)
NETWORK 37
	[L_R_Q] - LOW_R:R_TRIG(CLK: *) --- (LOW_R_Q)
NETWORK 38
	[LOW_R_Q]
		EN --- SUB(XH_SHU_OUT, 1) => XH_SHU_OUT
NETWORK 39
	*
		EN --- LE(XH_SHU_OUT, 0) => XH_SHU_0
NETWORK 40
	[HIGH_KA] - { [/XH_JT_KA] | [JT_KA] }
		EN --- MOVE(DWORD_TO_WORD(DIV(TIME_TO_DWORD(OPEN_ET), 1000))) => XH_T_XSH
NETWORK 41
	[LOW_KA]
		EN --- MOVE(DWORD_TO_WORD(DIV(TIME_TO_DWORD(CLOSE_ET), 1000))) => XH_T_XSH
NETWORK 42
	[XH_JT_KA] - [/JT_KA]
		EN --- MOVE(DWORD_TO_WORD(DIV(TIME_TO_DWORD(JT_OPEN_ET), 1000))) => XH_T_XSH
_END_LD_
(* the same logic as Structured Text *)
(* Network 1 *)
IF NOT TD_R OR WBKZL_IN OR GRD_ALA THEN
	XH_SHU_OUT := 0;
END_IF;
(* Network 2: see the listing above *)
(* Network 3 *)
XW := WD_IN - 600;
(* Network 4 *)
XQ_WD_OUT := XW + XQ_WD_XZH;
(* Network 5 *)
YL_WD(YL_IN := MNL_OUT * 10);
YL_T_OUT := YL_WD.YL_T;
(* Network 6 *)
GRD_OUT := XQ_WD_OUT - YL_T_OUT;
GRD_KA := GRD_OUT <= GRD_IN;
GRD_KA_0 := GRD_YSH_SET = 0;
(* Network 7 *)
GRD_OPEN(EN_IN := YSJ_IN AND GRD_KA AND NOT RESET AND NOT GRD_KA_0, TIME_IN := GRD_YSH_SET);
GRD_YSH_XSH := GRD_OPEN.ET_OUT;
GRD_ALA := (GRD_OPEN.OUT OR GRD_ALA) AND NOT GRD_KA_0 AND NOT RESET;
(* Network 8 *)
JQ_NJ_SHU_0 := JQ_NJ_SHU = 0;
(* Network 9 *)
JJQ_TOF(IN := NOT HIGH_KA, PT := T#10S);
JJQ_OUT := JJQ_TOF.Q AND KAIJI AND JQ_NJ_SHU_0 AND OPEN_IN;
(* Network 10 *)
MNL_OUT := REAL_TO_INT(MNL_R + INT_TO_REAL(MNL_XZH));
(* Network 11: see the listing above *)
(* Network 12: see the listing above *)
(* Network 13 *)
HIGH_KA := KAIJI AND (HIGH AND OPEN_IN OR HIGH_KA AND NOT MID_KA AND NOT LOW_KA) AND NOT LOW_KA AND OPEN_IN;
(* Network 14 *)
MID_KA := KAIJI AND MID AND NOT LOW_KA;
(* Network 15 *)
LOW_KA := KAIJI AND LOW OR NOT KAIJI OR WBKZL_IN OR NOT OPEN_IN AND TJ_ZHH_OUT;
(* Network 16 *)
IF LOW_KA THEN
	XH_ZHT := 0;
END_IF;
(* Network 17 *)
IF MID_KA THEN
	XH_ZHT := 1;
END_IF;
(* Network 18 *)
IF HIGH_KA THEN
	XH_ZHT := 2;
END_IF;
(* Network 19 *)
MID_R(CLK := MID_KA);
IF MID_R.Q THEN
	XH_SHU_OUT := JQ_NJ_SHU;
END_IF;
(* Network 20 *)
IF NOT TD_R THEN
	XH_SHU_OUT := 0;
END_IF;
(* Network 21 *)
JQ_OPEN_SET := DWORD_TO_TIME(WORD_TO_DWORD(JQ_OPEN_YSH) * 60000);
(* Network 22 *)
CLOSE_SET := DWORD_TO_TIME(WORD_TO_DWORD(CLOSE_YSH) * 1000);
(* Network 23 *)
OPEN_SET := DWORD_TO_TIME(WORD_TO_DWORD(OPEN_YSH) * 1000);
(* Network 24 *)
H_TON(IN := HIGH_KA AND NOT H_R_Q AND NOT XH_STOP AND XH_JD, PT := OPEN_SET);
OPEN_ET := H_TON.ET;
H_R_Q := H_TON.Q;
(* Network 25 *)
HIG_R(CLK := H_R_Q);
HIG_KA_R(CLK := HIGH_KA);
IF HIG_R.Q OR HIG_KA_R.Q THEN
	XH_SHU_OUT := XH_SHU_OUT + 1;
END_IF;
(* Network 26 *)
XH_JD := XH_NE_3 AND XH_NE_6 AND XH_NE_9 AND XH_NE_12 AND XH_NE_18 OR JT_KA;
(* Network 27 *)
XH_NE_3 := XH_SHU_OUT <> 3;
XH_NE_6 := XH_SHU_OUT <> 6;
XH_NE_9 := XH_SHU_OUT <> 9;
XH_NE_12 := XH_SHU_OUT <> 12;
XH_NE_18 := XH_SHU_OUT <> 18;
(* Network 28 *)
XH_EQ_3 := XH_SHU_OUT = 3;
XH_EQ_6 := XH_SHU_OUT = 6;
XH_EQ_9 := XH_SHU_OUT = 9;
XH_EQ_12 := XH_SHU_OUT = 12;
XH_EQ_15 := XH_SHU_OUT = 15;
XH_EQ_18 := XH_SHU_OUT = 18;
(* Network 29 *)
XH_SHU := BOOL_TO_WORD(XH_SHU_OUT >= 3) + BOOL_TO_WORD(XH_SHU_OUT >= 6) + BOOL_TO_WORD(XH_SHU_OUT >= 9) + BOOL_TO_WORD(XH_SHU_OUT >= 12) + BOOL_TO_WORD(XH_SHU_OUT >= 15) + BOOL_TO_WORD(XH_SHU_OUT >= 18);
(* Network 30 *)
JT_SHU := SEL(TD_R, 0, BOOL_TO_WORD(NOT JQ_1_BH_IN) + BOOL_TO_WORD(NOT JQ_2_BH_IN) + BOOL_TO_WORD(NOT JQ_3_BH_IN) + BOOL_TO_WORD(NOT JQ_4_BH_IN) + BOOL_TO_WORD(NOT JQ_5_BH_IN) + BOOL_TO_WORD(NOT JQ_6_BH_IN));
(* Network 31 *)
XH_STOP := XH_SHU >= JT_SHU;
(* Network 32 *)
IF XH_STOP THEN
	XH_SHU_OUT := JT_SHU * 3;
END_IF;
(* Network 33 *)
XH_JT_KA := XH_EQ_3 OR XH_EQ_6 OR XH_EQ_9 OR XH_EQ_12 OR XH_EQ_15;
(* Network 34 *)
JT_TON(IN := XH_JT_KA, PT := JQ_OPEN_SET);
JT_OPEN_ET := JT_TON.ET;
JT_KA := (JT_TON.Q OR JQ_A_OPEN_SET_0) AND (HIGH_KA OR MID_KA);
(* Network 35 *)
JQ_OPEN_SET_0 := JQ_OPEN_YSH = 0;
(* Network 36 *)
L_TON(IN := LOW_KA AND NOT XH_SHU_0 AND NOT L_R_Q, PT := CLOSE_SET);
CLOSE_ET := L_TON.ET;
L_R_Q := L_TON.Q;
(* Network 37 *)
LOW_R(CLK := L_R_Q);
LOW_R_Q := LOW_R.Q;
(* Network 38 *)
IF LOW_R_Q THEN
	XH_SHU_OUT := XH_SHU_OUT - 1;
END_IF;
(* Network 39 *)
XH_SHU_0 := XH_SHU_OUT <= 0;
(* Network 40 *)
IF HIGH_KA AND (NOT XH_JT_KA OR JT_KA) THEN
	XH_T_XSH := DWORD_TO_WORD(TIME_TO_DWORD(OPEN_ET) / 1000);
END_IF;
(* Network 41 *)
IF LOW_KA THEN
	XH_T_XSH := DWORD_TO_WORD(TIME_TO_DWORD(CLOSE_ET) / 1000);
END_IF;
(* Network 42 *)
IF XH_JT_KA AND NOT JT_KA THEN
	XH_T_XSH := DWORD_TO_WORD(TIME_TO_DWORD(JT_OPEN_ET) / 1000);
END_IF;
END_FUNCTION_BLOCK

(* POU JQ_NJ_SHU, LD *)
FUNCTION_BLOCK JQ_NJ_SHU
VAR_INPUT
	JQ_1_NJ: WORD;
	JQ_2_NJ: WORD;
	JQ_3_NJ: WORD;
	JQ_4_NJ: WORD;
	JQ_5_NJ: WORD;
	JQ_6_NJ: WORD;
	JQ_1_IN: BOOL;
	JQ_2_IN: BOOL;
	JQ_3_IN: BOOL;
	JQ_4_IN: BOOL;
	JQ_5_IN: BOOL;
	JQ_6_IN: BOOL;
END_VAR
VAR_OUTPUT
	JQ_NJ_ROM: WORD;
END_VAR
VAR
	JQ_1_NJ_ROM: WORD;
	JQ_2_NJ_ROM: WORD;
	JQ_3_NJ_ROM: WORD;
	JQ_4_NJ_ROM: WORD;
	JQ1: YSJ_NJ_SHU;
	JQ2: YSJ_NJ_SHU;
	JQ3: YSJ_NJ_SHU;
	JQ4: YSJ_NJ_SHU;
	JQ_5_NJ_ROM: WORD;
	JQ_6_NJ_ROM: WORD;
	JQ5: YSJ_NJ_SHU;
	JQ6: YSJ_NJ_SHU;
END_VAR
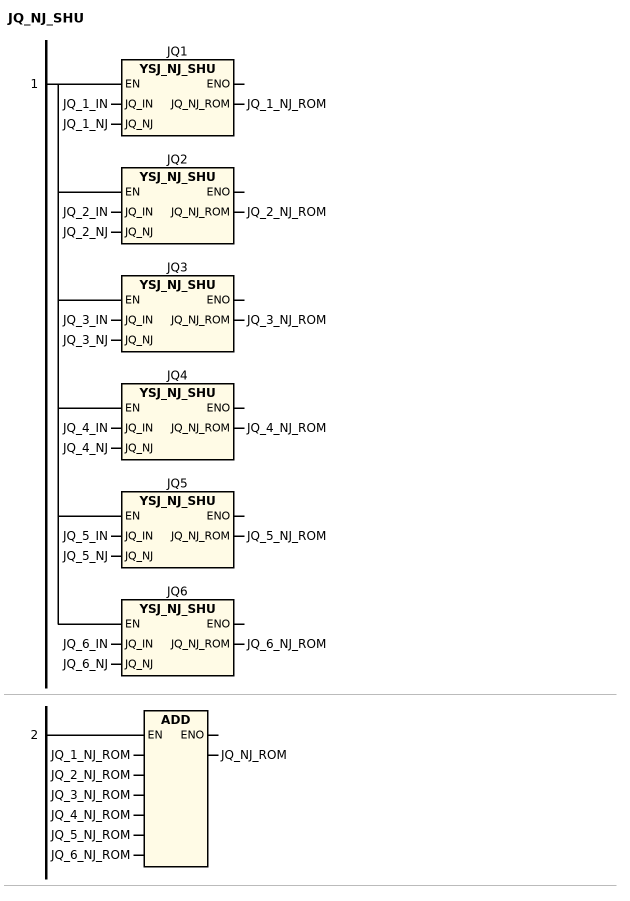
_LD_ (* Ladder Diagram *)
NETWORK 1
	*
		EN --- JQ1:YSJ_NJ_SHU(JQ_IN: JQ_1_IN, JQ_NJ: JQ_1_NJ) => JQ_1_NJ_ROM
		EN --- JQ2:YSJ_NJ_SHU(JQ_IN: JQ_2_IN, JQ_NJ: JQ_2_NJ) => JQ_2_NJ_ROM
		EN --- JQ3:YSJ_NJ_SHU(JQ_IN: JQ_3_IN, JQ_NJ: JQ_3_NJ) => JQ_3_NJ_ROM
		EN --- JQ4:YSJ_NJ_SHU(JQ_IN: JQ_4_IN, JQ_NJ: JQ_4_NJ) => JQ_4_NJ_ROM
		EN --- JQ5:YSJ_NJ_SHU(JQ_IN: JQ_5_IN, JQ_NJ: JQ_5_NJ) => JQ_5_NJ_ROM
		EN --- JQ6:YSJ_NJ_SHU(JQ_IN: JQ_6_IN, JQ_NJ: JQ_6_NJ) => JQ_6_NJ_ROM
NETWORK 2
	*
		EN --- ADD(JQ_1_NJ_ROM, JQ_2_NJ_ROM, JQ_3_NJ_ROM, JQ_4_NJ_ROM, JQ_5_NJ_ROM, JQ_6_NJ_ROM) => JQ_NJ_ROM
_END_LD_
(* the same logic as Structured Text *)
(* Network 1 *)
JQ1(JQ_IN := JQ_1_IN, JQ_NJ := JQ_1_NJ);
JQ_1_NJ_ROM := JQ1.JQ_NJ_ROM;
JQ2(JQ_IN := JQ_2_IN, JQ_NJ := JQ_2_NJ);
JQ_2_NJ_ROM := JQ2.JQ_NJ_ROM;
JQ3(JQ_IN := JQ_3_IN, JQ_NJ := JQ_3_NJ);
JQ_3_NJ_ROM := JQ3.JQ_NJ_ROM;
JQ4(JQ_IN := JQ_4_IN, JQ_NJ := JQ_4_NJ);
JQ_4_NJ_ROM := JQ4.JQ_NJ_ROM;
JQ5(JQ_IN := JQ_5_IN, JQ_NJ := JQ_5_NJ);
JQ_5_NJ_ROM := JQ5.JQ_NJ_ROM;
JQ6(JQ_IN := JQ_6_IN, JQ_NJ := JQ_6_NJ);
JQ_6_NJ_ROM := JQ6.JQ_NJ_ROM;
(* Network 2 *)
JQ_NJ_ROM := JQ_1_NJ_ROM + JQ_2_NJ_ROM + JQ_3_NJ_ROM + JQ_4_NJ_ROM + JQ_5_NJ_ROM + JQ_6_NJ_ROM;
END_FUNCTION_BLOCK

(* POU YSJ_NJ_SHU, LD *)
FUNCTION_BLOCK YSJ_NJ_SHU
VAR_INPUT
	JQ_IN: BOOL;
	JQ_NJ: WORD;
END_VAR
VAR_OUTPUT
	JQ_NJ_ROM: WORD;
END_VAR
VAR
END_VAR
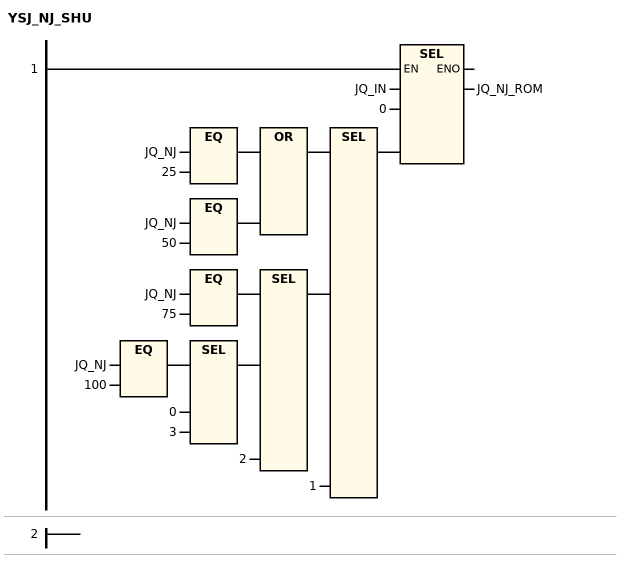
_LD_ (* Ladder Diagram *)
NETWORK 1
	*
		EN --- SEL(JQ_IN, 0, SEL(OR(EQ(JQ_NJ, 25), EQ(JQ_NJ, 50)), SEL(EQ(JQ_NJ, 75), SEL(EQ(JQ_NJ, 100), 0, 3), 2), 1)) => JQ_NJ_ROM
NETWORK 2
	*
_END_LD_
(* the same logic as Structured Text *)
(* Network 1 *)
JQ_NJ_ROM := SEL(JQ_IN, 0, SEL((JQ_NJ = 25) OR (JQ_NJ = 50), SEL(JQ_NJ = 75, SEL(JQ_NJ = 100, 0, 3), 2), 1));
(* Network 2 *)
END_FUNCTION_BLOCK

(* POU YL_WD, LD *)
FUNCTION_BLOCK YL_WD
VAR_INPUT
	YL_IN: INT;
END_VAR
VAR_OUTPUT
       YL_T: INT;
END_VAR
VAR
	YT_41_50: INT;
	YT_31_40: INT;
	YT_11_20: INT;
	YT_1_10: INT;
	YT_9_0: INT;
	YT_19_10: INT;
	YT_29_20: INT;
	YL_IN_R: REAL;
	YL_T_KA: INT;
	YT_51_60: INT;
	YT_41_31: INT;
END_VAR
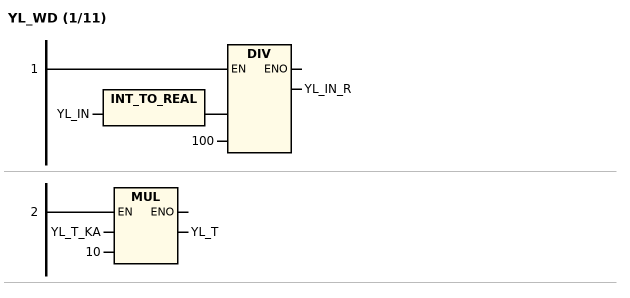
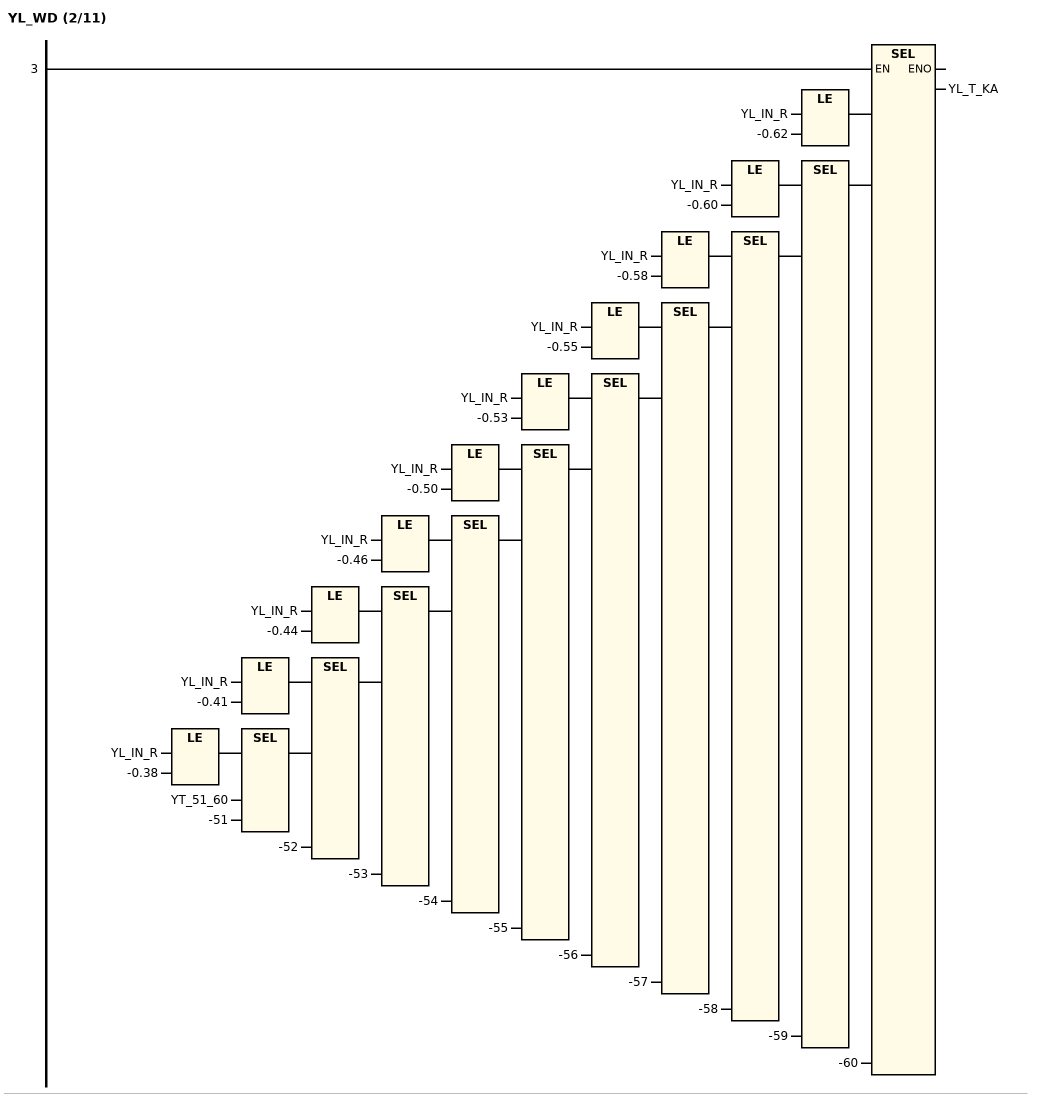
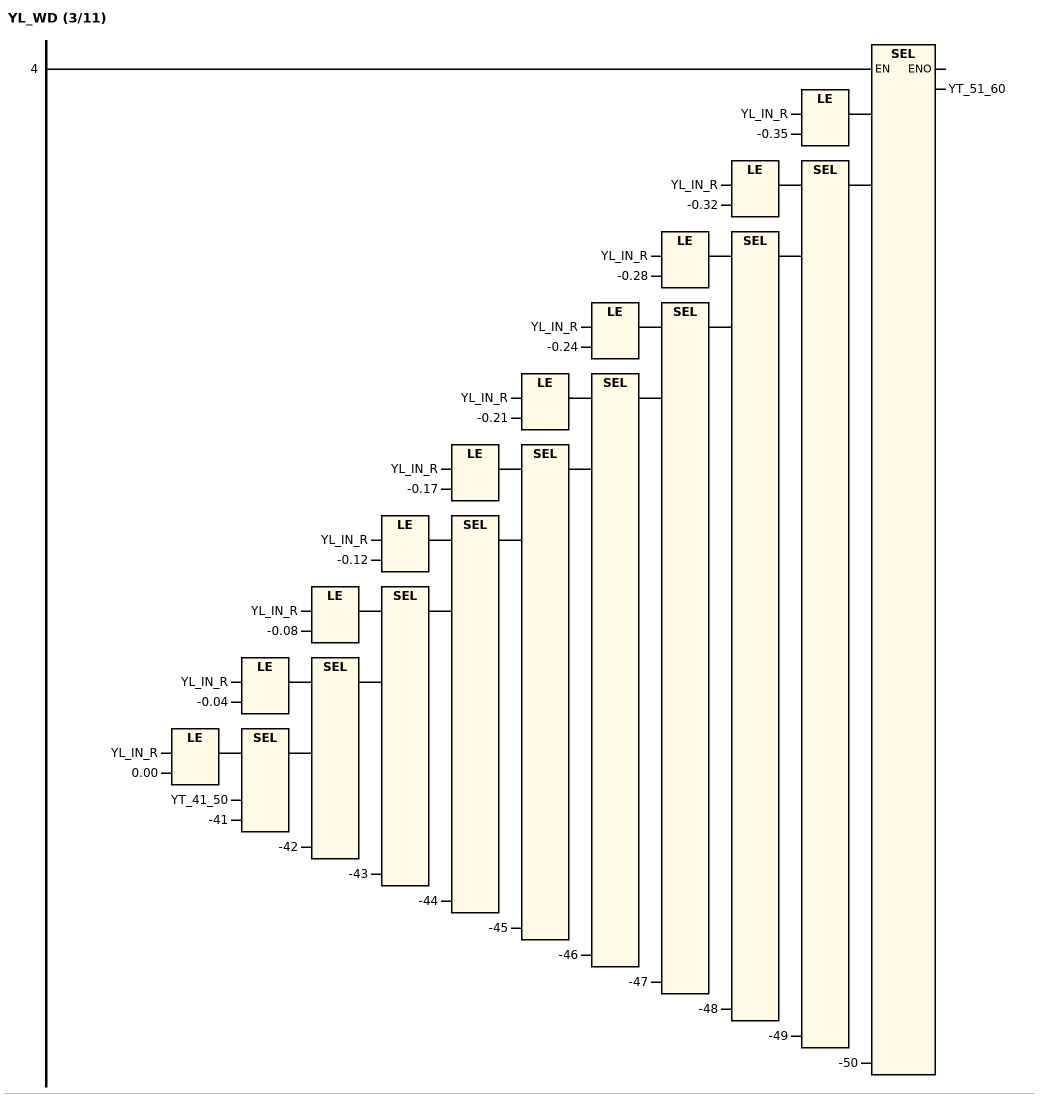
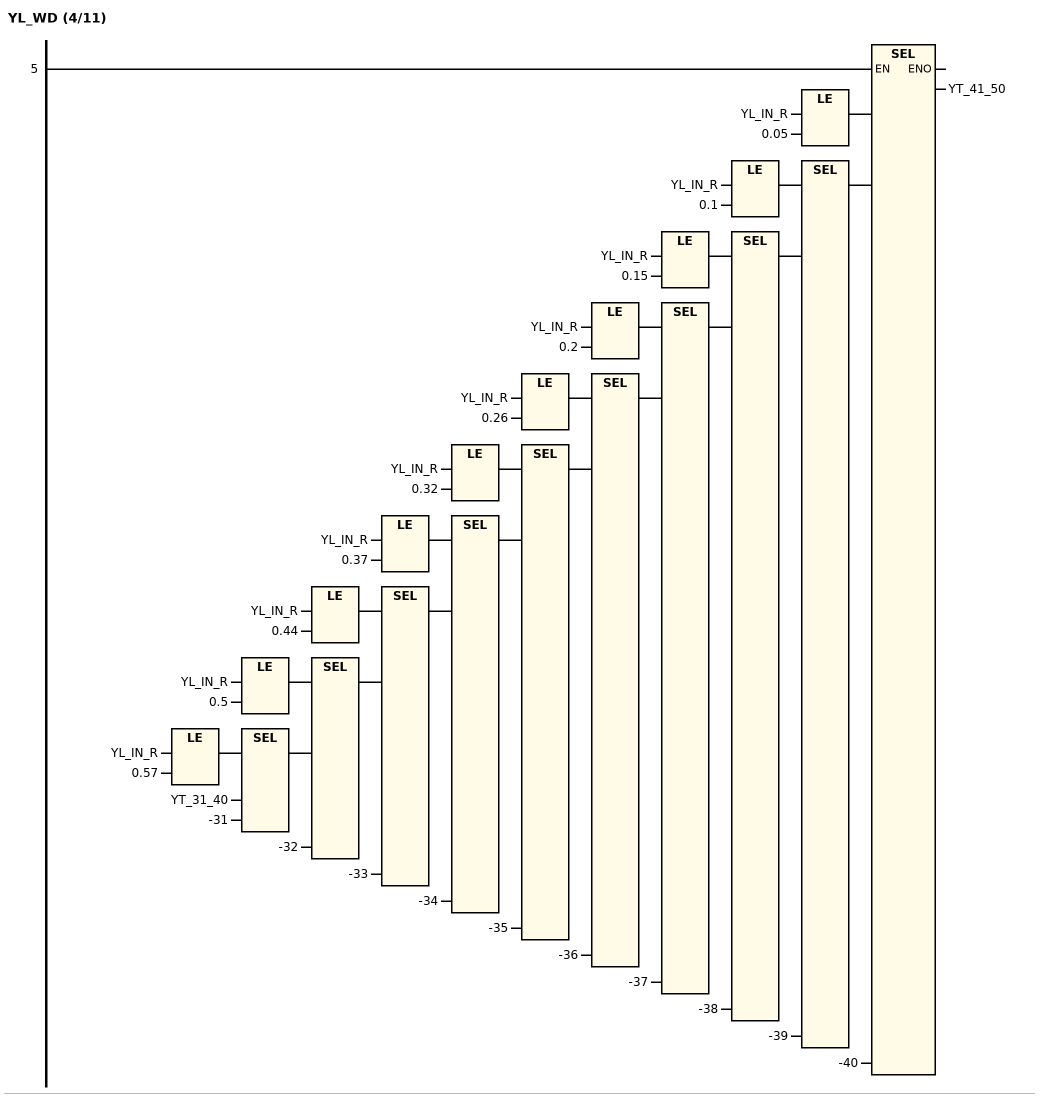
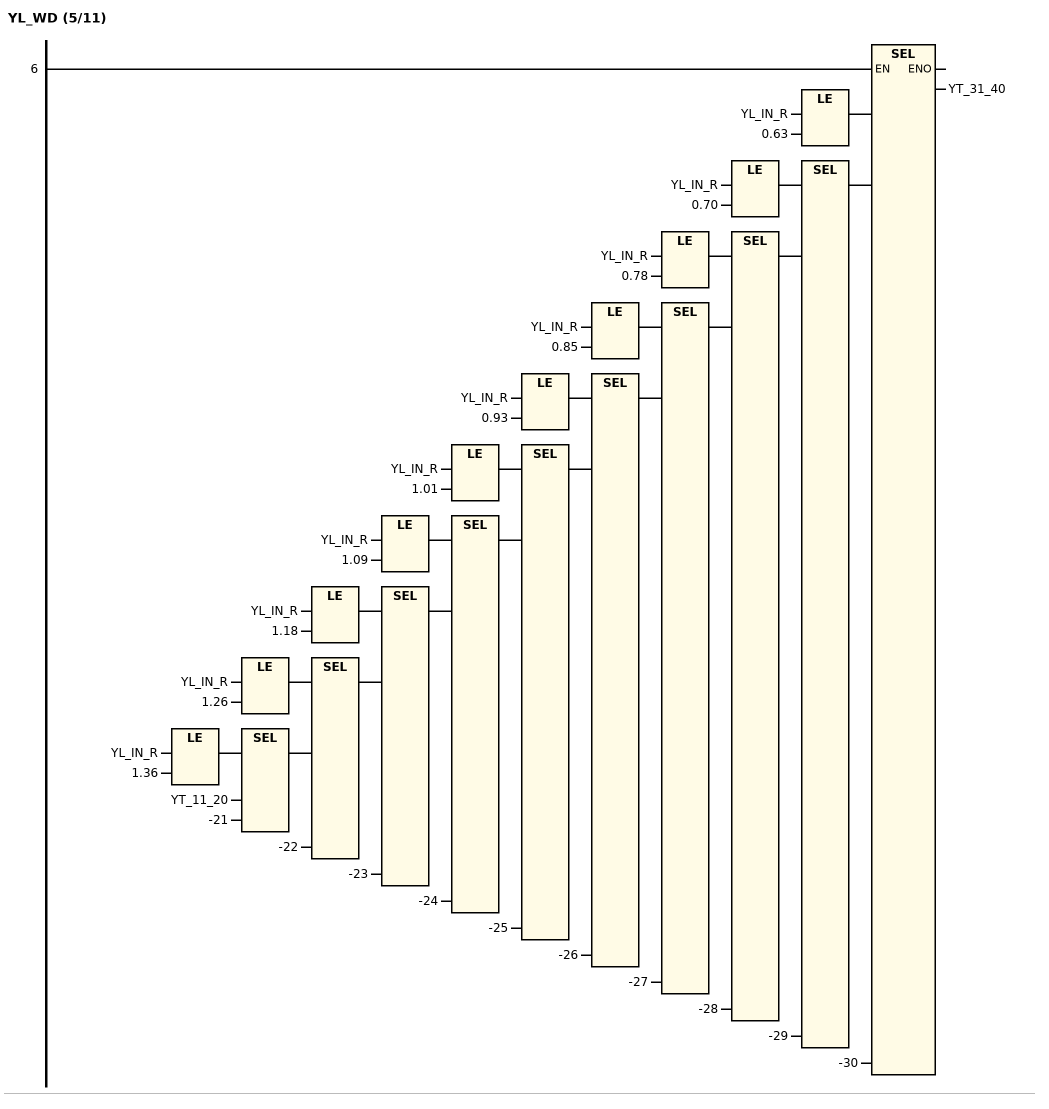
